{attribute 'qualified_only'}
VAR_GLOBAL
END_VAR

(* stored: Version 1.1.0.1, ProductVersion 3.1.4022.7
   GVL GVL_06_Output_Servo_Motor_Shelf_C: Id {51d68d2c-e408-4ffc-97c7-64fe2d0d72a6} *)
